PROGRAM prgComEffIO
VAR
	fbCom			: FB_MqttCommunicator;
END_VAR

fbCom(
	bConnect:= TRUE, 
	sUserName:= 'e4244e14-25de-4873-b6c5-796d986e1983', 
	sUserPassword:= '91460717-fd5f-4424-8478-e62b11d57fc5', 
	eSavePositionCertificate:= eSavePositionOnPLC.ePostionHardDisk, 
	bConnected=> , 
	bError=> , 
	hrErrorCode=> , 
	eConnectionState=> , 
	eErrorMessage_Out=> );

END_PROGRAM

(* stored: Version 1.1.0.1, ProductVersion 3.1.4024.9
   POU prgComEffIO: Id {229bd226-3c0c-4816-823a-75063aeb2d03}, SpecialFunc None *)
